Fanuc KAREL source: ko00046.KL

PROGRAM KO00046
%STACKSIZE=65535
%PRIORITY=65535
%NOLOCKGROUP
VAR
P1 : POSITION
P2 : JOINTPOS9
F : BOOLEAN
OUT : XYZWPR
BEGIN
F=TRUE
-- UNSAFE_SOURCE_IR line 11: OUT = MIRROR(convert_position_to_xyzwprext(P1), convert_jointpos9_to_position(P2), F)
END KO00046
